{attribute 'GeneratedUsingTerminal: KL9900-0064'}
{attribute addProperty BoxType "KL9900-0064"}
{attribute addProperty Id "Channel_1AT %Q*Channel_0F0CD9400"}
{attribute addProperty CRC "573031259"}
{attribute addProperty Size "0"}
TYPE KL_2227C35B :
STRUCT
	{attribute addProperty Name "Channel_1"}
	Channel_1 : Channel_0F0CD940;
END_STRUCT
END_TYPE

(* stored: Version 1.2.0.0, ProductVersion 3.1.4024.9
   DUT KL_2227C35B: Id {adc34d9e-604c-4429-bea4-fee41dc5150b} *)
